FUNCTION_BLOCK FB_Vehiculo
VAR_INPUT
	velocidad : REAL;
END_VAR
VAR_OUTPUT
END_VAR
VAR
END_VAR

METHOD getVelocidad : REAL
VAR_INPUT
END_VAR
getVelocidad := velocidad;
END_METHOD

END_FUNCTION_BLOCK

(* stored: Version 1.1.0.1, ProductVersion 3.1.4024.12
   POU FB_Vehiculo: Id {bebaaf0e-1adc-4bbd-8b5c-f9bacc7f4ae8}, SpecialFunc None
   Method getVelocidad: Id {eecfef92-45e0-446c-90fd-ee4f150246fb} *)
